# EPICS IOC start-up script: test/startup/st.ymir-mcs1.iocsh
require ethercatmc,USER

epicsEnvSet("MOTOR_PORT",    "$(SM_MOTOR_PORT=MCU1)")
epicsEnvSet("IPADDR",        "$(SM_IPADDR=10.102.10.44)")
epicsEnvSet("IPPORT",        "$(SM_IPPORT=48898)")
epicsEnvSet("AMSNETIDIOC",   "$(SM_AMSNETID=10.102.10.49.1.1)")
epicsEnvSet("ASYN_PORT",     "$(SM_ASYN_PORT=MC_CPU1)")
epicsEnvSet("PREFIX",        "$(SM_PREFIX=YMIR-)")
epicsEnvSet("PREC",          "$(SM_PREC=3)")
epicsEnvSet("ECM_NUMAXES",     "9")
epicsEnvSet("ECM_OPTIONS",   "adsPort=852;amsNetIdRemote=10.102.10.44.1.1;amsNetIdLocal=$(AMSNETIDIOC)")

epicsEnvSet("ECM_MOVINGPOLLPERIOD", "0")
epicsEnvSet("ECM_IDLEPOLLPERIOD",   "0")

< ethercatmcController.iocsh

#
# AXIS 1
#
epicsEnvSet("AXISCONFIG",      "")
epicsEnvSet("AXIS_NAME",      "$(SM_AXIS_NAME=HvSht:MC-Pne-01)")
epicsEnvSet("AXIS_NO",         "$(SM_AXIS_NO=1)")
< ethercatmcShutter.iocsh

#
# AXIS 2
#
epicsEnvSet("AXISCONFIG",      "")
epicsEnvSet("AXIS_NAME",      "$(SM_AXIS_NAME=Fil:MC-Pne-01)")
epicsEnvSet("AXIS_NO",         "$(SM_AXIS_NO=2)")
< ethercatmcShutter.iocsh

#
# AXIS 3
#
epicsEnvSet("AXISCONFIG",      "")
epicsEnvSet("AXIS_NAME",      "$(SM_AXIS_NAME=Fil:MC-Pne-02)")
epicsEnvSet("AXIS_NO",         "$(SM_AXIS_NO=3)")
< ethercatmcShutter.iocsh

#
# AXIS 4
#
epicsEnvSet("AXISCONFIG",      "")
epicsEnvSet("AXIS_NAME",      "$(SM_AXIS_NAME=Spare-AXIS-1)")
epicsEnvSet("AXIS_NO",         "$(SM_AXIS_NO=4)")
epicsEnvSet("RAWENCSTEP_ADEL", 0)
epicsEnvSet("RAWENCSTEP_MDEL", 0)
< ethercatmcIndexerAxis.iocsh
< ethercatmcAxisdebug.iocsh

#
# AXIS 5
#
epicsEnvSet("AXISCONFIG",      "")
epicsEnvSet("AXIS_NAME",      "$(SM_AXIS_NAME=Spare-AXIS-2)")
epicsEnvSet("AXIS_NO",         "$(SM_AXIS_NO=5)")
epicsEnvSet("RAWENCSTEP_ADEL", 0)
epicsEnvSet("RAWENCSTEP_MDEL", 0)
< ethercatmcIndexerAxis.iocsh
< ethercatmcAxisdebug.iocsh

#
# AXIS 6
#
epicsEnvSet("AXISCONFIG",      "")
epicsEnvSet("AXIS_NAME",      "$(SM_AXIS_NAME=ColSl1:MC-SlYp-01)")
epicsEnvSet("AXIS_NO",         "$(SM_AXIS_NO=6)")
epicsEnvSet("RAWENCSTEP_ADEL", 0)
epicsEnvSet("RAWENCSTEP_MDEL", 0)
< ethercatmcIndexerAxis.iocsh
< ethercatmcAxisdebug.iocsh

#
# AXIS 7
#
epicsEnvSet("AXISCONFIG",      "")
epicsEnvSet("AXIS_NAME",      "$(SM_AXIS_NAME=ColSl1:MC-SlYm-01)")
epicsEnvSet("AXIS_NO",         "$(SM_AXIS_NO=7)")
epicsEnvSet("RAWENCSTEP_ADEL", 0)
epicsEnvSet("RAWENCSTEP_MDEL", 0)
< ethercatmcIndexerAxis.iocsh
< ethercatmcAxisdebug.iocsh

#
# AXIS 8
#
epicsEnvSet("AXISCONFIG",      "")
epicsEnvSet("AXIS_NAME",      "$(SM_AXIS_NAME=ColSl1:MC-SlZp-01)")
epicsEnvSet("AXIS_NO",         "$(SM_AXIS_NO=8)")
epicsEnvSet("RAWENCSTEP_ADEL", 0)
epicsEnvSet("RAWENCSTEP_MDEL", 0)
< ethercatmcIndexerAxis.iocsh
< ethercatmcAxisdebug.iocsh

#
# AXIS 9
#
epicsEnvSet("AXISCONFIG",      "")
epicsEnvSet("AXIS_NAME",      "$(SM_AXIS_NAME=ColSl1:MC-SlZm-01)")
epicsEnvSet("AXIS_NO",         "$(SM_AXIS_NO=9)")
epicsEnvSet("RAWENCSTEP_ADEL", 0)
epicsEnvSet("RAWENCSTEP_MDEL", 0)
< ethercatmcIndexerAxis.iocsh
< ethercatmcAxisdebug.iocsh

epicsEnvSet("MOVINGPOLLPERIOD", "9")
epicsEnvSet("IDLEPOLLPERIOD",   "100")
ethercatmcStartPoller("$(MOTOR_PORT)", "$(MOVINGPOLLPERIOD)", "$(IDLEPOLLPERIOD)")
